INTERFACE PUBLIC StoppingCommands EXTENDS ClearedStateCommands, ActionStateCommands

END_INTERFACE

(* stored: Version 1.1.0.1, ProductVersion 3.1.4026.18
   Itf StoppingCommands: Id {28886706-ab5d-0d83-1519-135622573c5d} *)
